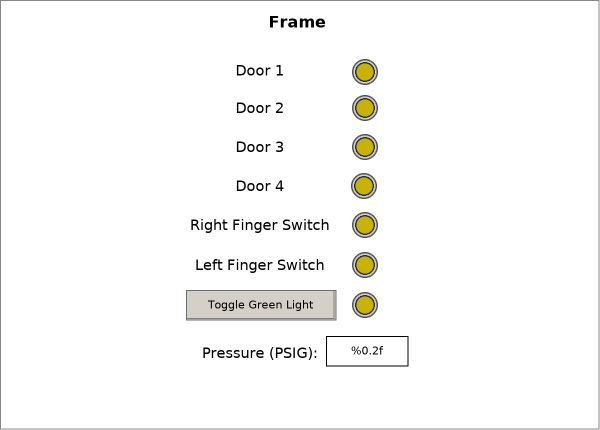
VISUALIZATION Manual_Frame  // 600x430
    Label (0,7 600x30), "Frame"
    Label (185,57 150x27), "Door 1"
    Label (185,93 150x30), "Door 2"
    Label (185,132 150x30), "Door 3"
    Label (185,210 150x30), "Right Finger Switch"
    Label (185,250 150x30), "Left Finger Switch"
    Lamp1 (350,57 30x30), variable: MAIN.Frame.diDoor1, style: Lamp-Lamp1-Yellow
    Lamp1 (350,93 30x30), variable: MAIN.Frame.diDoor2, style: Lamp-Lamp1-Yellow
    Lamp1 (350,132 30x30), variable: MAIN.Frame.diDoor3, style: Lamp-Lamp1-Yellow
    Lamp1 (350,210 30x30), variable: MAIN.Frame.diControlLeft, style: Lamp-Lamp1-Yellow
    Lamp1 (350,250 30x30), variable: MAIN.Frame.diControlRight, style: Lamp-Lamp1-Yellow
    Lamp1 (350,290 30x30), variable: MAIN.Frame.doGreen, style: Lamp-Lamp1-Yellow
    Button (186,290 150x30), "Toggle Green Light"
        OnMouseClick: execute { MAIN.Frame.GreenLight := NOT MAIN.Frame.GreenLight; }
    Label (185,338 150x30), "Pressure (PSIG):"
    Rectangle (326,336 82x30), "%0.2f", text variable: MAIN.Frame._pressure
    Label (185,171 150x30), "Door 4"
    Lamp1 (349,171 30x30), variable: MAIN.Frame.diDoor4, style: Lamp-Lamp1-Yellow
END_VISUALIZATION

(* stored: Version 1.1.0.1, ProductVersion 3.1.4024.9
   Visu Manual_Frame: Id {bbf353e5-63c8-4e99-8d50-66701cc07798} *)
